FUNCTION_BLOCK FB_Spring EXTENDS FB_SeasonBase
VAR_INPUT
END_VAR
VAR_OUTPUT
END_VAR
VAR
END_VAR

METHOD ChangeToSummerTyres
VAR_INPUT
END_VAR
THIS^._nTyresType := 1;
Tc2_System.ADSLOGSTR(msgCtrlMask := THIS^._nLogLevel,
                     msgFmtStr := 'Changed to summer tyres',
                     strArg := '');
END_METHOD

METHOD FB_init : BOOL
VAR_INPUT
    bInitRetains:           BOOL; // if TRUE, the retain variables are initialized (warm start / cold start)
    bInCopyCode:            BOOL;  // if TRUE, the instance afterwards gets moved into the copy code (online change)
    ipStateMachine:         I_StateMachine;
    ipParentObject:         I_Object;
END_VAR
THIS^._eState := E_Season.Spring;
END_METHOD

METHOD  NextSeason
VAR_INPUT
END_VAR
THIS^.ipStateMachine.SetState(THIS^.ipSeasonCtrl.StateSummer);
END_METHOD

METHOD OnEntry
VAR_INPUT
END_VAR
SUPER^.OnEntry();
THIS^._bWindBlowing     := FALSE;
THIS^._bRaining         := TRUE;
THIS^._bSunShining      := FALSE;
THIS^._bSnowing         := TRUE;
THIS^._nLeavesState     := 1;
END_METHOD

METHOD OnExit
SUPER^.OnExit();
THIS^._bWindBlowing     := FALSE;
THIS^._bRaining         := FALSE;
THIS^._bSunShining      := FALSE;
THIS^._bSnowing         := TRUE;
THIS^._nLeavesState     := 1;
END_METHOD

END_FUNCTION_BLOCK

(* stored: Version 1.1.0.1, ProductVersion 3.1.4024.12
   POU FB_Spring: Id {3921a95a-def8-4684-80c2-5c5aa3716243}, SpecialFunc None
   Method ChangeToSummerTyres: Id {a3e93717-ff32-4f39-ba65-b3a10ce5f0da}
   Method FB_init: Id {c8139c82-1b18-43cd-855a-a86968a34c9f}
   Method NextSeason: Id {111fa8b5-fd58-47a9-99dd-562d52a5e48b}
   Method OnEntry: Id {d6b5dffe-3a55-4d85-8bc2-153cb570d300}
   Method OnExit: Id {6cb36855-ee1a-4ca1-aee7-e15d7b3c7943} *)
